{attribute 'GeneratedUsingTerminal: EL3783-0000-0018'}
{attribute addProperty BoxType "EL3783-0000-0018"}
{attribute addProperty Id "I2_SamplesAT %I*I2_Samples_1109DCAA40"}
{attribute addProperty CRC "1126159308"}
{attribute addProperty Size "40"}
TYPE L2_Current_Samples_431FD3CC EXTENDS InputBase_8311D824 :
STRUCT
	{attribute addProperty Name "I2_Samples"}
	I2_Samples AT %I* : I2_Samples_1109DCAA;
END_STRUCT
END_TYPE

(* stored: Version 1.2.0.0, ProductVersion 3.1.4024.9
   DUT L2_Current_Samples_431FD3CC: Id {f4ab052f-df8e-464c-8319-1f1b99940db8} *)
